(* IEC 61131-3 sources: beckhoffAutomationInterface/ST/Shark/App/Shark/Functions, 5 files *)

(* ---- F_GetBeckhoffTempChannelConfig.st ---- *)
(* Resolves the COMPLETE per-channel controller configuration for one heat channel.

   This is the single boundary between the GVL config tables and the temperature
   subsystem: FB_TemperatureSubsystem consumes the returned struct instead of
   reaching into GVL_TemperatureZoneConfig itself (DIP).

   It composes the per-zone template (F_GetBeckhoffTempZoneConfig) and layers the
   per-channel specialisation on top: identity, single-authority enable policy,
   per-channel PID gains, and per-channel duty-cycle cap.

   (Mirror of the PRO function. Shark has no safety thermocouple, so that
   PRO block is intentionally absent here.)

   Returns sZoneID = 'INVALID' for an out-of-range / unpopulated zone. *)
FUNCTION F_GetBeckhoffTempChannelConfig : ST_BeckhoffTempZoneConfig
VAR_INPUT
    eZone          : E_HeatZone;   // 1..CONTROLLABLE_ZONE_MAX
    nGlobalIdx     : INT;          // 1..CHANNEL_MAX (flat channel index)
    nChannelInZone : INT;          // 1..nChannelCount (position within the zone)
END_VAR
VAR
    stConfig : ST_BeckhoffTempZoneConfig;
    fDuty    : LREAL;
END_VAR
    // Zone-level template: setpoint clamp, output limits, timing, ramp.
    stConfig := F_GetBeckhoffTempZoneConfig(eZone := eZone);
    IF stConfig.sZoneID = 'INVALID' THEN
        F_GetBeckhoffTempChannelConfig := stConfig;
        RETURN;
    END_IF

    // The ZONE is the single control authority — channels must never self-enable;
    // enable/disable always cascades from FB_HeatZone.
    stConfig.bAutoEnable := FALSE;

    // Per-channel identity for error traceability, e.g. 'HETR_HEAD_E1'.
    stConfig.sZoneID := CONCAT(TO_STRING(eZone), CONCAT('_E', TO_STRING(nChannelInZone)));

    // Per-channel maximum duty cycle (hardware-rated cap): used as the controller
    // output limit AND as a clamp on the autotune step, so a channel can never
    // exceed its rating, even while tuning.
    IF nGlobalIdx >= 1 AND nGlobalIdx <= GVL_TemperatureZones.CHANNEL_MAX THEN
        fDuty := GVL_TemperatureZoneConfig.MAX_DUTY_CYCLE[nGlobalIdx];
        stConfig.rOutputMax := fDuty;
        stConfig.stControllerParams.fYMax := fDuty;
        IF stConfig.stControllerParams.fYTuneHeating > fDuty THEN
            stConfig.stControllerParams.fYTuneHeating := fDuty;
        END_IF
    END_IF

    // Per-channel PID gains. Channels in a zone are physically distinct bands
    // and may each have their own tuned gains (autotune results live here).
    IF nGlobalIdx >= 1 AND nGlobalIdx <= GVL_TemperatureZones.CHANNEL_MAX THEN
        stConfig.stExternalPID.KpHeat := GVL_TemperatureZoneConfig.PID_GAINS[nGlobalIdx].rKp;
        stConfig.stExternalPID.TnHeat := GVL_TemperatureZoneConfig.PID_GAINS[nGlobalIdx].tTn;
        stConfig.stExternalPID.TvHeat := GVL_TemperatureZoneConfig.PID_GAINS[nGlobalIdx].tTv;
        stConfig.stExternalPID.TdHeat := GVL_TemperatureZoneConfig.PID_GAINS[nGlobalIdx].tTd;
    END_IF

    F_GetBeckhoffTempChannelConfig := stConfig;
END_FUNCTION

(* ---- F_GetBeckhoffTempZoneConfig.st ---- *)
(* Returns zone-specific configuration directly. *)
FUNCTION F_GetBeckhoffTempZoneConfig : ST_BeckhoffTempZoneConfig
VAR_INPUT
    eZone : E_HeatZone;
END_VAR
VAR
    stConfig : ST_BeckhoffTempZoneConfig;
    stParams : ST_CTRL_TempCtrlParameter;
    stZoneConfig : ST_TemperatureZoneConfig;
END_VAR

    IF eZone < 1 OR eZone > GVL_TemperatureZones.CONTROLLABLE_ZONE_MAX THEN
        stConfig.sZoneID := 'INVALID';
        F_GetBeckhoffTempZoneConfig := stConfig;
        RETURN;
    END_IF

    stZoneConfig := GVL_TemperatureZoneConfig.ZONE_CONFIG[eZone];

    // Skip unpopulated zones
    IF NOT stZoneConfig.bPopulated THEN
        stConfig.sZoneID := 'INVALID';
        F_GetBeckhoffTempZoneConfig := stConfig;
        RETURN;
    END_IF

    // Zone limits and safety thresholds
    stConfig.rMinSetpoint := stZoneConfig.rMinSetpoint;
    stConfig.rMaxSetpoint := stZoneConfig.rMaxSetpoint;

    // Dynamic safety limit: Zone Max + Margin (e.g. 400 + 10 = 410)
    stConfig.rSafetyMaxTemp := stZoneConfig.rMaxSetpoint + GVL_TemperatureSystem.TEMP_SAFETY_MARGIN;
    stConfig.rAbsoluteMaxTemp := stZoneConfig.rMaxSetpoint + GVL_TemperatureSystem.TEMP_ABSOLUTE_MARGIN;

    stConfig.rSetpointTolerance := GVL_TemperatureSystem.CTRL_SETPOINT_TOLERANCE;
    stConfig.tMaxContinuousOn := GVL_TemperatureSystem.CTRL_MAX_CONTINUOUS_ON;
    stConfig.rOutputMin := GVL_TemperatureSystem.OUTPUT_MIN;
    stConfig.rOutputMax := GVL_TemperatureSystem.OUTPUT_MAX;
    stConfig.rOutputSafeDefault := GVL_TemperatureSystem.OUTPUT_SAFE_DEFAULT;

    // Controller mode and failure behavior
    stParams.iMode := E_CTRL_ControlMode.eCTRL_ControlMode_HEATING;
    stParams.iReactionOnFailure := E_CTRL_ReactionOnFailure.eCTRL_ReactionOnFailure_StopController;
    stParams.bSelCtrlParameterSet := TRUE;
    stParams.dwAlarmSupp := GVL_TemperatureSystem.CTRL_ALARM_SUPPRESSION;

    // Timing configuration
    stParams.tCtrlCycleTime := GVL_TemperatureSystem.CTRL_CYCLE_TIME;
    stParams.tTaskCycleTime := GVL_TemperatureSystem.CTRL_TASK_CYCLE_TIME;

    // Auto-tuning parameters
    stParams.iTuningMode := E_CTRL_TuneMode.eCTRL_TuneMode_HEATING;
    stParams.tTuneStabilisation := GVL_TemperatureSystem.CTRL_TUNE_STABILIZATION;
    stParams.fEndTunePercentHeating := GVL_TemperatureSystem.TUNE_END_PERCENT_HEATING;
    stParams.fYTuneHeating := GVL_TemperatureSystem.TUNE_Y_HEATING;
    stParams.fYStableHeating := GVL_TemperatureSystem.TUNE_Y_STABLE;
    stParams.fScalingFactor := GVL_TemperatureSystem.CTRL_SCALING_FACTOR;

    // Ramping configuration
    stParams.bEnableSoftStart := TRUE;
    stParams.bEnableRamping := TRUE;
    stParams.fWVeloPos := F_RampRateToVelocity(stZoneConfig.rHeatingRampRate);
    stParams.fWVeloNeg := F_RampRateToVelocity(stZoneConfig.rCoolingRampRate);

    // Output limits
    stParams.fYMin := GVL_TemperatureSystem.OUTPUT_MIN;
    stParams.fYMax := GVL_TemperatureSystem.OUTPUT_MAX;
    stParams.fYManual := GVL_TemperatureSystem.OUTPUT_MANUAL_DEFAULT;
    stParams.fYOnFailure := GVL_TemperatureSystem.OUTPUT_SAFE_DEFAULT;

    // PWM configuration
    stParams.tPWMCycleTime := GVL_TemperatureSystem.CTRL_PWM_CYCLE_TIME;
    stParams.tPWMMinOffTime := GVL_TemperatureSystem.CTRL_PWM_MIN_TIME;
    stParams.tPWMMinOnTime := GVL_TemperatureSystem.CTRL_PWM_MIN_TIME;

    stParams.iControllerType := E_CTRL_ControllerType.eCTRL_ControllerType_PID;

    // Alarm thresholds (relative to setpoint)
    stParams.TempLow := GVL_TemperatureSystem.ALARM_TEMP_LOW;
    stParams.TempLowLow := GVL_TemperatureSystem.ALARM_TEMP_LOW_LOW;
    stParams.TempHigh := GVL_TemperatureSystem.ALARM_TEMP_HIGH;
    stParams.TempHighHigh := GVL_TemperatureSystem.ALARM_TEMP_HIGH_HIGH;
    stParams.TempAbsoluteHigh := GVL_TemperatureSystem.SENSOR_MAX_TEMP;
    stParams.TempAbsoluteLow := GVL_TemperatureSystem.SENSOR_MIN_RANGE;

    // PID tuning multipliers
    stParams.fTuneKp := GVL_TemperatureSystem.TUNE_KP;
    stParams.fTuneTn := GVL_TemperatureSystem.TUNE_TN;
    stParams.fTuneTv := GVL_TemperatureSystem.TUNE_TV;
    stParams.fTuneTd := GVL_TemperatureSystem.TUNE_TD;

    // Setpoint limits
    stParams.fWMin := stZoneConfig.rMinSetpoint;
    stParams.fWMax := stZoneConfig.rMaxSetpoint;

    // NOTE: PID gains (stExternalPID) are NOT set here. They are per-channel and
    // applied in F_GetBeckhoffTempChannelConfig from GVL_TemperatureZoneConfig.PID_GAINS.

    stConfig.stControllerParams := stParams;
    stConfig.sZoneID := TO_STRING(eZone);

    F_GetBeckhoffTempZoneConfig := stConfig;
END_FUNCTION

(* ---- F_GetCompany.st ---- *)
FUNCTION F_GetCompany : STRING(80)
VAR
END_VAR
    F_GetCompany := 'ATLANT 3D';
END_FUNCTION

(* ---- F_GetHeatZoneConfig.st ---- *)
(* Builds an ST_HeatZoneConfig from the per-zone row in GVL_TemperatureZoneConfig.
   Used by FB_TemperatureSubsystem when initialising each FB_HeatZone. *)
FUNCTION F_GetHeatZoneConfig : ST_HeatZoneConfig
VAR_INPUT
    eZone : E_HeatZone;
END_VAR
VAR
    stConfig     : ST_HeatZoneConfig;
    stZoneConfig : ST_TemperatureZoneConfig;
END_VAR

    IF eZone < 1 OR eZone > GVL_TemperatureZones.CONTROLLABLE_ZONE_MAX THEN
        stConfig.sZoneID := 'INVALID';
        F_GetHeatZoneConfig := stConfig;
        RETURN;
    END_IF

    stZoneConfig := GVL_TemperatureZoneConfig.ZONE_CONFIG[eZone];

    IF NOT stZoneConfig.bPopulated THEN
        stConfig.sZoneID := 'INVALID';
        F_GetHeatZoneConfig := stConfig;
        RETURN;
    END_IF

    stConfig.sZoneID    := TO_STRING(eZone);
    stConfig.eAggregation := stZoneConfig.eAggregation;
    stConfig.rMaxDeltaWarn := stZoneConfig.rMaxDeltaWarn;
    stConfig.rMaxDeltaTrip := stZoneConfig.rMaxDeltaTrip;
    stConfig.rMinSetpoint := stZoneConfig.rMinSetpoint;
    stConfig.rMaxSetpoint := stZoneConfig.rMaxSetpoint;

    F_GetHeatZoneConfig := stConfig;
END_FUNCTION

(* ---- F_GetTitle.st ---- *)
FUNCTION F_GetTitle : STRING(80)
VAR
END_VAR
    F_GetTitle := 'PLC_SHARK_PROJ';
END_FUNCTION
